FUNCTION "FPC_MAPPING" : Bool
{ S7_Optimized_Access := 'FALSE' }
AUTHOR : FESTO
FAMILY : 'E-DRIVE'
VERSION : 4.1
   VAR_INPUT
      Mode : Bool;
   END_VAR

   VAR_IN_OUT
      FML_REF : "t_DT_FML_REF";
   END_VAR

   VAR_TEMP
      _Word : Word;
      BByte2 AT _Word : Array[1..2] of Byte;
      _DINT : DInt;
      BByte4 AT _DINT : Array[1..4] of Byte;
      Req_Identifier : Int;
      Resp_Identifier : Int;
   END_VAR


BEGIN
	(*############################################################
	   FESTO AG  Co., Esslingen
	   Copyright (c) 2015. All rights reserved.

	   NAME OF FUNCTION BLOCK:         FPC_MAPPING
	   VERSION NUMBER:                 V4.1
	   COMPOSER:                       bejk

	   -----------------------------------------------------
	   Date        Name                Activity
	   06.08.2015  Benjamin Kilgus     created (V1.0)
	   29.08.2016  Benjamin Klein      version changed (V4.1)

	############################################################*)

	(* MAP INPUTS *)
	IF NOT #Mode THEN

	  // Byte1 FPCS
	  #FML_REF.FPCS_Modus := SHR(IN := (#FML_REF.InData.FPC[1] AND 2#11110000), N := 4);

	  // decoding of EFPC modus
	  CASE BYTE_TO_INT(#FML_REF.FPCS_Modus) OF
	    0: (* old style *)
	    (*
	    -------------- Byte 1 --------------- Byte 2 ---------------------- Byte 3/4 ------------------- Byte 5..8 ----
	    |  8  7  6  5  4  |  3  2  1  0  |              | 15 14 13 12 |  11  | 10 9 8 7 6 5 4 3 2 1 0 |               |
	    |    FPCS Modus   |     res      |   Subindex   |      AK     |  SPM |        PNU             |     Value     |
	    ---------------------------------------------------------------------------------------------------------------
	    AK:  Response Identifier (Antwortkennung)
	    SPM: NOT used
	    PNU: Parameternummer / Parameter-Number
	    *)
	      // Byte1
	        // zero in this CASE
	      // Byte2
	        #FML_REF.ActSubindex := #FML_REF.InData.FPC[2];

	      // Byte3/4
	      #BByte2[1] := #FML_REF.InData.FPC[3];
	      #BByte2[2] := #FML_REF.InData.FPC[4];
	      #Resp_Identifier := WORD_TO_INT(SHR(IN := (#_Word AND 2#1111000000000000), N := 12));
	      #FML_REF.ActPNU := #_Word AND 2#0000011111111111;

	      // Byte 5..8 parameter value
	      #BByte4[1] := #FML_REF.InData.FPC[5];
	      #BByte4[2] := #FML_REF.InData.FPC[6];
	      #BByte4[3] := #FML_REF.InData.FPC[7];
	      #BByte4[4] := #FML_REF.InData.FPC[8];
	      #FML_REF.ParamValueRD := #_DINT;

	    1, 2, 3:(* modus: 1 = PNU extended; 2 = KO; 3 = CAN Objects *)
	    (*
	    -------------- Byte 1 --------------- Byte 2 ------------------- Byte 3/4----------------- Byte 5..8 ----
	    |   7  6  5  4  |  3  2  1  0  |              | 15 14 13 12 11 10 9 8 7 6 5 4 3 2 1 0 |               |
	    |  FPCS Modus   |     AK       |   Subindex   |   PNU extended or KO or CAN Object    |     Value     |
	    -------------------------------------------------------------------------------------------------------
	    AK:  Response Identifier (Antwortkennung)
	    *)

	      // Byte 1 FPCS
	      #Resp_Identifier := WORD_TO_INT(#FML_REF.InData.FPC[1] AND 2#00001111);

	      // Byte 2 Subindex
	      #FML_REF.ActSubindex := #FML_REF.InData.FPC[2];

	      // Byte 3+4 **PKE/ PNU/ KO/ CAN**
	      #BByte2[1] := #FML_REF.InData.FPC[3];
	      #BByte2[2] := #FML_REF.InData.FPC[4];
	      #FML_REF.ActPNU := #_Word;

	      // Byte 5..8 parameter value
	      #BByte4[1] := #FML_REF.InData.FPC[5];
	      #BByte4[2] := #FML_REF.InData.FPC[6];
	      #BByte4[3] := #FML_REF.InData.FPC[7];
	      #BByte4[4] := #FML_REF.InData.FPC[8];
	      #FML_REF.ParamValueRD := #_DINT;

	  4,5:(* FPCS_Modus 4=Parameter File; 5=Firmware File *)
	  (*
	  ------ BYTE 1 ------------|-- BYTE 2 -|--BYTE 3..8 ---|
	  | 7  6  5  4 | 3  2  1  0 |           |               |
	  | FPCS Modus |   res      | Packet-ID |  6 BYTE Data  |
	  -------------------------------------------------------
	    Packet-ID: -------------- BYTE 2 ----------
	               | 7    6    5  | 4  3  2  1  0 |
	               | Control Bits |   Sequence-Nr |
	               --------------------------------
	 *)
	  // Byte 1 FPCS
	  #Resp_Identifier := WORD_TO_INT(#FML_REF.InData.FPC[1] AND 2#00001111);
	  #FML_REF.RespID := #Resp_Identifier;

	  //---- Byte 2 Packet-ID ----
	  #FML_REF.FPCS_Packet.BitSequenceNr := WORD_TO_INT(#FML_REF.InData.FPC[2] AND 2#00011111);
	  #FML_REF.FPCS_Packet.Control := WORD_TO_INT(SHR(IN := (#FML_REF.InData.FPC[2] AND 2#11100000), N := 5));
	  //---- Byte 3..8 Data ----
	  #FML_REF.FPCS_Packet.Data[1] := #FML_REF.InData.FPC[3];
	  #FML_REF.FPCS_Packet.Data[2] := #FML_REF.InData.FPC[4];
	  #FML_REF.FPCS_Packet.Data[3] := #FML_REF.InData.FPC[5];
	  #FML_REF.FPCS_Packet.Data[4] := #FML_REF.InData.FPC[6];
	  #FML_REF.FPCS_Packet.Data[5] := #FML_REF.InData.FPC[7];
	  #FML_REF.FPCS_Packet.Data[6] := #FML_REF.InData.FPC[8];


	    ELSE (* not implemented *)
	      #FPC_MAPPING := FALSE; (* Execution was not correct *)
	      RETURN;
	  END_CASE;

	  CASE #Resp_Identifier OF
	    0:(* No Transmission*)
	      #FML_REF.Done := FALSE;
	      #FML_REF.Err := FALSE;
	      #FML_REF.ActPNU := 0;
	      #FML_REF.ActSubindex := 0;
	      #FML_REF.ParamValueRD := 0;

	    5: (*Transmission Done*)
	      #FML_REF.Done := true;
	      #FML_REF.Err := FALSE;

	    7:(* Transmission Failed*)
	      #FML_REF.Done := TRUE;
	      #FML_REF.Err := TRUE;

	    ELSE (* not specified*)
	      #FML_REF.Done := TRUE;
	      #FML_REF.Err := TRUE;
	  END_CASE;

	  #FPC_MAPPING := TRUE; (* Execution was correct *)
	  RETURN;

	(* MAP OUTPUTS *)
	ELSE


	  (* create request identifier *)
	  #Req_Identifier := #FML_REF.ReqID;

	  CASE BYTE_TO_INT(#FML_REF.FPCC_Modus) OF
	    0: (* old style *)
	    (*
	    -------------- Byte 1 --------------- Byte 2 ---------------------- Byte 3 --------------------- Byte 5..8 ----
	    |  8  7  6  5  4  |  3  2  1  0  |              | 15 14 13 12 |  11  | 10 9 8 7 6 5 4 3 2 1 0 |               |
	    |    FPCS Modus   |     res      |   Subindex   |      AK     |  SPM |        PNU             |     Value     |
	    ---------------------------------------------------------------------------------------------------------------
	    AK:  Request Identifier (Auftragskennung)
	    SPM: NOT used
	    PNU: Parameternummer / Parameter-Number
	    *)
	    (* Byte 1 *)
	      #FML_REF.OutData.FPC[1] := SHL(IN := #FML_REF.FPCC_Modus, N := 4);
	      (* Byte 2 Subindex *)
	      #FML_REF.OutData.FPC[2] := #FML_REF.Subindex;
	      (* Byte 3+4 *)
	      #_Word := SHL(IN := INT_TO_WORD(#Req_Identifier), N := 12) OR (#FML_REF.PNU AND 16#07_FF);

	      (* Byte 5..8 *)
	      #_DINT := #FML_REF.ParamValueWR;
	      #FML_REF.OutData.FPC[3] := #BByte2[1]; //Convert PKE to Byte
	      #FML_REF.OutData.FPC[4] := #BByte2[2];

	      (* Set Output DATA OF DRIVE *)
	      #FML_REF.OutData.FPC[5] := #BByte4[1]; //Convert PWE to Byte
	      #FML_REF.OutData.FPC[6] := #BByte4[2];
	      #FML_REF.OutData.FPC[7] := #BByte4[3];
	      #FML_REF.OutData.FPC[8] := #BByte4[4];

	    1, 2, 3:(* modus: 1 = PNU extended; 2 = KO; 3 = CAN Objects *)
	    (*
	    -------------- Byte 1 --------------- Byte 2 ------------------- Byte 3 ------------------ Byte 5..8 ----
	    |  8  7  6  5  4  |  3  2  1  0  |              | 15 14 13 12 11 10 9 8 7 6 5 4 3 2 1 0 |               |
	    |    FPCS Modus   |     AK       |   Subindex   |   PNU extended or KO or CAN Object    |     Value     |
	    ---------------------------------------------------------------------------------------------------------
	    AK:  Request Identifier (Auftragskennung)
	    *)
	    (* Byte 1 *)
	      #FML_REF.OutData.FPC[1] := WORD_TO_BYTE(SHL(IN := #FML_REF.FPCC_Modus, N := 4) OR INT_TO_WORD(#Req_Identifier));
	      (* Byte 2 Subindex *)
	      #FML_REF.OutData.FPC[2] := #FML_REF.Subindex;
	      (* Byte 3+4 *)
	      #_Word := #FML_REF.PNU;
	      (* Byte 5..8 *)
	      #_DINT := #FML_REF.ParamValueWR;
	      #FML_REF.OutData.FPC[3] := #BByte2[1]; //Convert PKE to Byte
	      #FML_REF.OutData.FPC[4] := #BByte2[2];

	      (* Set Output DATA OF DRIVE *)
	      #FML_REF.OutData.FPC[5] := #BByte4[1]; //Convert PWE to Byte
	      #FML_REF.OutData.FPC[6] := #BByte4[2];
	      #FML_REF.OutData.FPC[7] := #BByte4[3];
	      #FML_REF.OutData.FPC[8] := #BByte4[4];

	  4,5:(* FPCC_Modus 4=parameter file; 5=firmware file
	        |---------- byte 1 --------|-- byte 2 --|-- byte 3..8 ---|
	        | 7  6  5  4  | 3  2  1  0 |            |                |
	        |   FPCC modus |   res      | packet-ID  |  6 byte data  |
	        ---------------------------------------------------------
	        Packet-ID:  | 7    6    5  | 4  3  2  1  0  |
	                    | control bits |  sequence-nr   |
	                    --------------------------------- *)
	       //---- byte 1 ----
	       #FML_REF.OutData.FPC[1] := WORD_TO_BYTE(SHL(IN := #FML_REF.FPCC_Modus, N := 4) OR INT_TO_WORD(#Req_Identifier));
	       //----byte 2 packet-ID ----
	       #FML_REF.OutData.FPC[2] := (SHL(IN := INT_TO_BYTE(#FML_REF.FPCC_Packet.Control), N := 5) OR (INT_TO_BYTE(#FML_REF.FPCC_Packet.BitSequenceNr) AND 16#1F));
	       //---- byte 3..8 data ----
	       #FML_REF.OutData.FPC[3] :=       #FML_REF.FPCC_Packet.Data[1];         // byte swapping for modbus data
	       #FML_REF.OutData.FPC[4] :=       #FML_REF.FPCC_Packet.Data[2];
	       #FML_REF.OutData.FPC[5] :=       #FML_REF.FPCC_Packet.Data[3];
	       #FML_REF.OutData.FPC[6] :=       #FML_REF.FPCC_Packet.Data[4];
	       #FML_REF.OutData.FPC[7] :=       #FML_REF.FPCC_Packet.Data[5];
	       #FML_REF.OutData.FPC[8] :=       #FML_REF.FPCC_Packet.Data[6];

	    ELSE (* not implemented *)
	      #FPC_MAPPING := FALSE; (* Execution was not correct *)
	      RETURN;
	END_CASE;

	  #FPC_MAPPING := TRUE; (* Execution was correct *)
	END_IF;

END_FUNCTION

